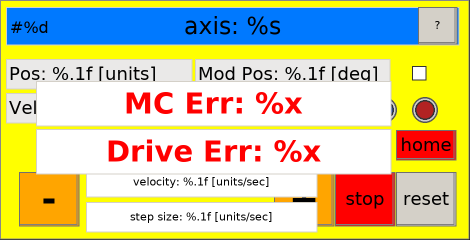
VISUALIZATION vis_Axis_Jog  // 470x240
VAR_IN_OUT
	Axis: ST_Axis;
END_VAR
VAR
	iBackGround_Description: INT;
END_VAR
    Rectangle (0,0 470x240), colour toggle: Axis.bEnabled
    Rectangle (0,0 470x240), colour toggle: Axis.bHomeDone AND Axis.bEnabled, invisible if: NOT Axis.bHomeDone
    Rectangle (0,0 470x240), colour toggle: Axis.bError, invisible if: Axis.bPowerOnN AND NOT Axis.bError
    Button (19,172 60x54), "-", colour toggle: Axis.bPowerOnN=0
        tap Axis.bJogBw
    Button (274,172 60x54), "+", colour toggle: Axis.bPowerOnP=0
        tap Axis.bJogFw
    Button (49,130 62x30), "Slow", colour toggle: Axis.eJogMode=MC_JOGMODE_STANDARD_SLOW
        OnMouseClick: execute { Axis.eJogMode:=MC_JOGMODE_STANDARD_SLOW; }
    Button (111,130 62x30), "Fast", colour toggle: Axis.eJogMode=MC_JOGMODE_STANDARD_FAST
        OnMouseClick: execute { Axis.eJogMode:=MC_JOGMODE_STANDARD_FAST; }
    Button (173,130 62x30), "Continous", colour toggle: Axis.eJogMode=MC_JOGMODE_CONTINOUS
        OnMouseClick: execute { Axis.eJogMode:=MC_JOGMODE_CONTINOUS; }
    Button (235,130 62x30), "Inching", colour toggle: Axis.eJogMode=MC_JOGMODE_INCHING
        OnMouseClick: execute { Axis.eJogMode:=MC_JOGMODE_INCHING; }
    Group (86,167 180x65)
        Textfield (0,0 231x30), "velocity: %.1f [units/sec]", text variable: Axis.fJogVelocity, invisible if: Axis.eJogMode<MC_JOGMODE_CONTINOUS
            OnMouseClick: write the text variable via Default, min 0, max 600
        Textfield (0,35 231x30), "step size: %.1f [units/sec]", text variable: Axis.fJogStep, invisible if: Axis.eJogMode<MC_JOGMODE_INCHING
            OnMouseClick: write the text variable via Default, min 0
    Group (6,59 187x64)
        Textfield (0,0 186x30), "Pos: %.1f [units]", text variable: Axis.fActPos
        Textfield (0,34 186x30), "Vel: %.1f [units/s]", text variable: Axis.fActVelo
    Textfield (6,7 453x38), "axis: %s", text variable: Axis.sAxis_Name
    Button (335,172 60x54), "stop"
        tap Axis.bStop
    Button (297,130 62x30), "Modulo", colour toggle: Axis.eJogMode=MC_JOGMODE_INCHING_MODULO
        OnMouseClick: execute { Axis.eJogMode:=MC_JOGMODE_INCHING_MODULO; }
    Textfield (7,11 50x33), "#%d", text variable: Axis.sAxis_Num
    Textfield (195,59 195x30), "Mod Pos: %.1f [deg]", tooltip "Modulo Position", text variable: Axis.fActPosModulo
    Label (195,94 67x30), "Power"
    DipSwitch (255,95 30x30), variable: Axis.bPowerOn, behaviour: TOGGLE, style: Switch-DipSwitch-Red
    Lamp1 (293,95 30x30), tooltip "Enabled", variable: Axis.bEnabled, style: Lamp-Lamp1-Green
    Button (396,130 60x30), "home", colour toggle: Axis.bHomeDone
        tap Axis.bHome
    Lamp1 (331,95 30x30), tooltip "Home sensor", variable: Axis.bHomeSen, style: Lamp-Lamp1-Yellow
    Button (396,172 60x54), "reset", colour toggle: Axis.bError
        tap Axis.bReset
    Lamp1 (369,95 30x30), tooltip "Home Done", variable: Axis.bHomeDone, style: Lamp-Lamp1-Blue
    Lamp1 (410,95 30x30), tooltip "Axis Error", variable: Axis.bError, style: Lamp-Lamp1-Red
    Frame (500,50 280x171), invisible if: iBackGround_Description=0
        shows vis_Axis_Control_Backgroud_Descripton()
        p3560616238: iBackGround_Description
    Button (418,7 39x37), "?"
        OnMouseClick: execute {
            IF iBackGround_Description<0 THEN;
            	iBackGround_Description:=0;
            ELSE;
            	iBackGround_Description:=-400;
            END_IF
        }
    Textfield (36,129 355x45), "Drive Err: %x", text variable: Axis.iErrorDI, invisible if: NOT Axis.bError
    Textfield (36,81 355x45), "MC Err: %x", text variable: Axis.Status.ErrorID, invisible if: NOT Axis.bError
    Checkbox (410,58 30x30), tooltip "Home mode Direct", variable: Axis.bHomeMode_Direct, invisible if: prg_User.actUser<4 AND Axis.bHomeMode_Direct=0
END_VISUALIZATION

(* stored: Version 1.1.0.1, ProductVersion 3.1.4024.12
   Visu vis_Axis_Jog: Id {6e1f0898-be79-4ca4-aa2c-81508d03f74c} *)
